(*
    This test-suite runs several asserts with the same parameters (same expected, actual, message) in the same cycle
    and in the same test.
    The reason we want the framework to support this is that theoretically the user could want to do an assert with the
    same message, in the same test, with the same data values for both expected and actual, although the data that the
    user does the assert on might be from different data sets.
*)
FUNCTION_BLOCK FB_MultipleAssertWithSameParametersInSameCycleWithSameTest EXTENDS TcUnit.FB_TestSuite

Assert_SeveralTimes();

METHOD PRIVATE Assert_SeveralTimes
VAR
    a : DWORD := 16#12345678;
    b : DWORD := 16#90ABCDEF;

    c : DWORD := 16#12345678;
    d : DWORD := 16#90ABCDEF;

    e : DWORD := 16#12345678;
    f : DWORD := 16#90ABCDEF;
END_VAR
TEST('Assert_SeveralTimes');

AssertEquals_DWORD(Expected := a,
                   Actual := b,
                   Message := 'Values differ');

AssertEquals_DWORD(Expected := c,
                   Actual := d,
                   Message := 'Values differ');

AssertEquals_DWORD(Expected := e,
                   Actual := f,
                   Message := 'Values differ');

TEST_FINISHED();
END_METHOD

END_FUNCTION_BLOCK

(* stored: Version 1.1.0.1, ProductVersion 3.1.4022.18
   POU FB_MultipleAssertWithSameParametersInSameCycleWithSameTest: Id {9957a11f-d554-4b5d-be35-f56d53aab4f2}, SpecialFunc None
   Method Assert_SeveralTimes: Id {cd07d59b-c5ef-4bab-a334-9a8ba622ccca} *)
